{attribute 'qualified_only'}
{attribute 'strict'}
TYPE LoadCaseType :
(
	VERY_LIGHT := 0, 
	LIGHT := 1, 
	MEDIUM := 2, 
	MODERATELY_HEAVY := 3, 
	HEAVY := 4
);
END_TYPE

(* stored: Version 1.1.0.1, ProductVersion 3.1.4024.12
   DUT LoadCaseType: Id {402cb31e-d666-4d3b-8afd-e0efe8e7de06} *)
